(* Logix 5000 project; controller R5_CSS vendor 1 type 14 code 74 rev 19.11; software revision 19.01; part 8 of 20 *)
(* tags used below, declared in another part *)
   Const_CubicInchToGal : REAL;
   FC101 : FLOW_CONTROL;   // QUENCH BASIN FLOW TRANSMITTER CONTROL
   FC101_PIDE : PID_ENHANCED;
   FC140 : FLOW_CONTROL;
   FC140_DIFF_FT : REAL;
   FC140A : FLOW_CONTROL;   // QUENCH TOWER UPPER SPRAY FLOW CONTROL
   FC140A_FT_Pcnt : REAL;
   FC140B : FLOW_CONTROL;   // QUENCH TOWER LOWER SPRAY FLOW CONTROL
   FC140B_FT_Pcnt : REAL;
   FCV410 : ValveControl_TwoWay;
   FCV410_AUTO_ONS : BOOL;
   FCV410_ClosedMinSP : DINT;
   FCV410_ClosedTON : TIMER;
   FCV410_HoldDelaySecSP : DINT;
   FCV410_HoldDelayTOF : TIMER;
   FCV410_LT_Hold : BOOL;
   FCV410_MANUAL_ONS : BOOL;
   FCV410_On : BOOL;
   FCV410_Open : BOOL;
   FCV410_OpenSecSP : DINT;
   FCV410_OpenTON : TIMER;
   FireFlowAlarm_ONS2 : BOOL;
   FireFlowAlarm_SetLC101 : BOOL;
   FireFlowAlarmFromUTL : BOOL;
   FT140_Ratio : REAL;
   FT140_TOTAL_FLOW : REAL;
   H3_LC101 : LEVEL_CONTROL;
   HX401A : PUMP_CONTROL;   // HEAT EXCHANGER A
   HX401A_QI_AUTO_OS : BOOL;
   HX401A_QI_MAN_OS : BOOL;
   HX401B : PUMP_CONTROL;   // HEAT EXCHANGER B
   HX401B_QI_AUTO_OS : BOOL;
   HX401B_QI_MAN_OS : BOOL;
   LC101 : LEVEL_CONTROL;   // QUENCH TOWER BASIN LIT
   LC101_AUTO_ONS1 : BOOL;
   LC101_LAHH_MaxTime_TMR : TIMER;
   LC101_LAHH_MaxTimeAlm : BOOL;
   LC101_LAHH_MaxTimeMinSP : REAL;
   LC101_LT_Temp : REAL;
   LC101_MANUAL_ONS1 : BOOL;
   LC101_PIDE : PID_ENHANCED;
   LC101_PIDE_AUTO : BOOL;
   LC101_PIDE_CV_Hold : REAL;
   LC205 : LEVEL_CONTROL;   // OVERHEAD CONDENSER BASIN LEVEL CONTROL
   LC205_Totalize_Calc : BOOL;
   LC205_Totalize_End : REAL;
   LC205_Totalize_Gal : REAL;
   LC205_Totalize_Inches : REAL;
   LC205_Totalize_Ini : BOOL;
   LC205_Totalize_Start : REAL;
   LC205_Totalize_TOF : TIMER;
   LC205_Totalize_Vessel1_Diameter_inches : REAL;
   LC205_Totalize_Vessel1_Gal : REAL;
   LC205_Totalize_Vessel1_Rad_inches : REAL;
   LC205_Totalize_Vessel2_Diameter_inches : REAL;
   LC205_Totalize_Vessel2_Gal : REAL;
   LC205_Totalize_Vessel2_Rad_inches : REAL;
   LC303A : LEVEL_CONTROL;   // AQUEOUS PHASE OF PRIMARY SETTLER
   MV361 : ValveControl_TwoWay;
   MV361_AUTO_ONS1 : BOOL;
   MV361_Open : BOOL;
   ONE_SHOT : BOOL[32];
   P101A : PUMP_CONTROL;
   P101B : PUMP_CONTROL;
   P205 : PUMP_CONTROL;   // OVERHEAD CONDENSER TRANSFER PUMP
   P205_START_ONS : BOOL;
   P205_STOP_ONS : BOOL;
   PID1_TCV101 : PID;
   PID_TCV101_TON : TIMER;
   QuenchFlowMeterFailed : BOOL;
   TIMER : TIMER[50];   // HX A TIMER FOR START
   TMR_FAULT : DINT;
(* MainProgram, continued *)

ROUTINE FCV410_BasinLevelHotWaterFlushValve   (* ladder *)
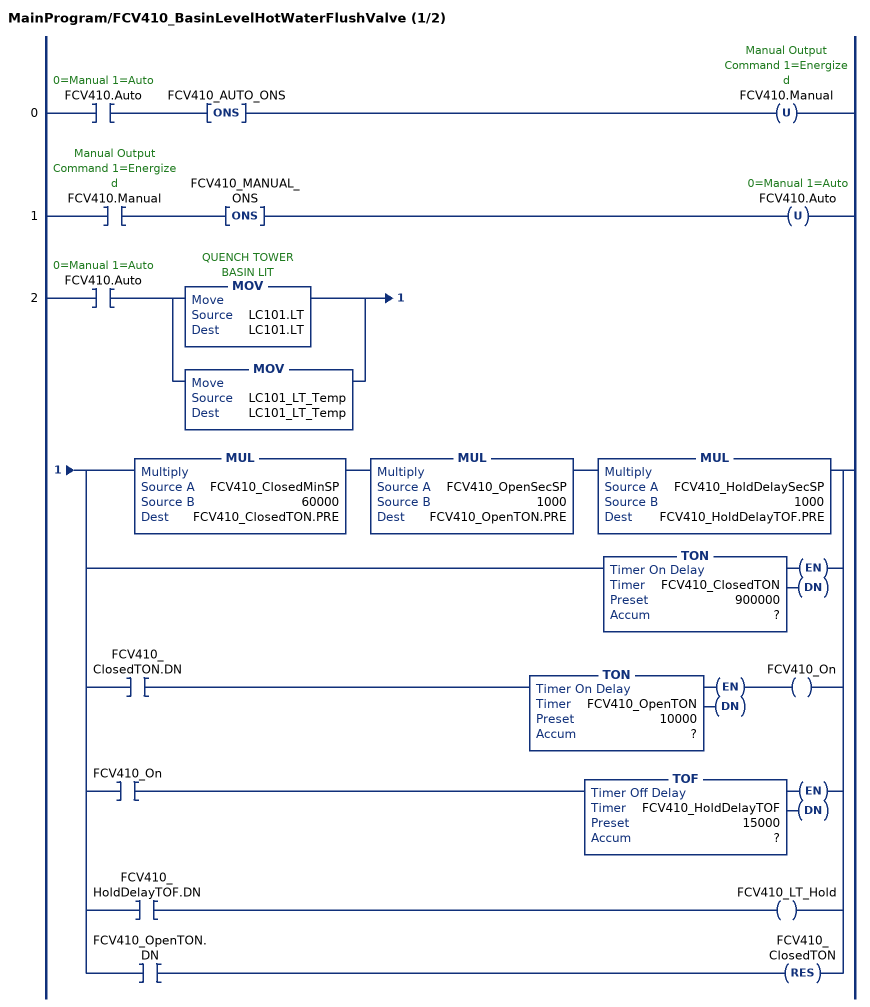
   0: XIC(FCV410.Auto)ONS(FCV410_AUTO_ONS)OTU(FCV410.Manual);
   1: XIC(FCV410.Manual)ONS(FCV410_MANUAL_ONS)OTU(FCV410.Auto);
   2: XIC(FCV410.Auto)[MOV(LC101.LT,LC101.LT) ,MOV(LC101_LT_Temp,LC101_LT_Temp) ][MUL(FCV410_ClosedMinSP,60000,FCV410_ClosedTON.PRE) MUL(FCV410_OpenSecSP,1000,FCV410_OpenTON.PRE) MUL(FCV410_HoldDelaySecSP,1000,FCV410_HoldDelayTOF.PRE) ,TON(FCV410_ClosedTON,?,?) ,XIC(FCV410_ClosedTON.DN) TON(FCV410_OpenTON,?,?) OTE(FCV410_On) ,XIC(FCV410_On) TOF(FCV410_HoldDelayTOF,?,?) ,XIC(FCV410_HoldDelayTOF.DN) OTE(FCV410_LT_Hold) ,XIC(FCV410_OpenTON.DN) RES(FCV410_ClosedTON) ];
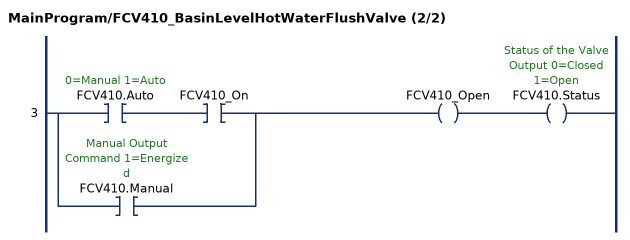
   3: [XIC(FCV410.Auto) XIC(FCV410_On) ,XIC(FCV410.Manual) ]OTE(FCV410_Open)OTE(FCV410.Status);
END_ROUTINE

ROUTINE FT140_QuenchFlowDelta   (* ladder *)
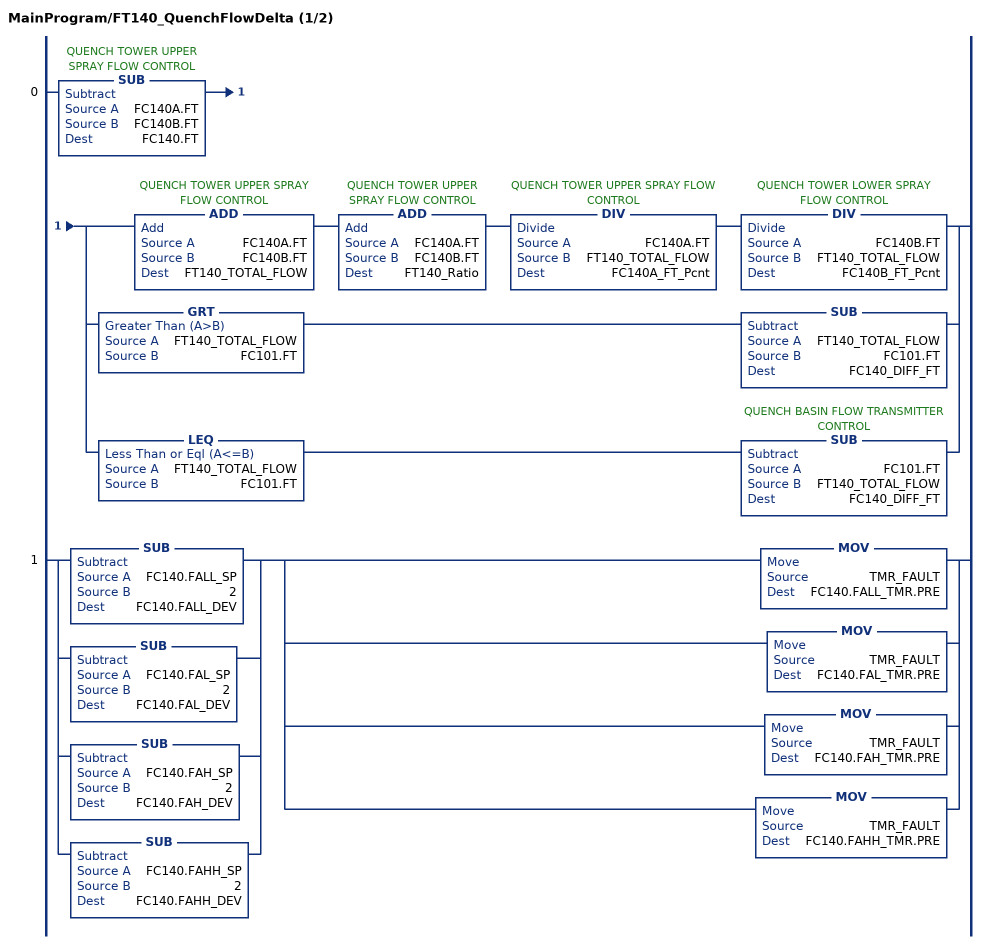
   0: SUB(FC140A.FT,FC140B.FT,FC140.FT)[ADD(FC140A.FT,FC140B.FT,FT140_TOTAL_FLOW) ADD(FC140A.FT,FC140B.FT,FT140_Ratio) DIV(FC140A.FT,FT140_TOTAL_FLOW,FC140A_FT_Pcnt) DIV(FC140B.FT,FT140_TOTAL_FLOW,FC140B_FT_Pcnt) ,GRT(FT140_TOTAL_FLOW,FC101.FT) SUB(FT140_TOTAL_FLOW,FC101.FT,FC140_DIFF_FT) ,LEQ(FT140_TOTAL_FLOW,FC101.FT) SUB(FC101.FT,FT140_TOTAL_FLOW,FC140_DIFF_FT) ];
   1: [SUB(FC140.FALL_SP,2,FC140.FALL_DEV) ,SUB(FC140.FAL_SP,2,FC140.FAL_DEV) ,SUB(FC140.FAH_SP,2,FC140.FAH_DEV) ,SUB(FC140.FAHH_SP,2,FC140.FAHH_DEV) ][MOV(TMR_FAULT,FC140.FALL_TMR.PRE) ,MOV(TMR_FAULT,FC140.FAL_TMR.PRE) ,MOV(TMR_FAULT,FC140.FAH_TMR.PRE) ,MOV(TMR_FAULT,FC140.FAHH_TMR.PRE) ];
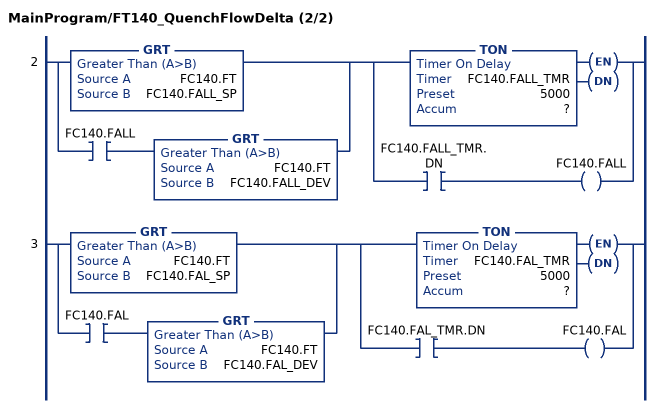
   2: [GRT(FC140.FT,FC140.FALL_SP) ,XIC(FC140.FALL) GRT(FC140.FT,FC140.FALL_DEV) ][TON(FC140.FALL_TMR,?,?) ,XIC(FC140.FALL_TMR.DN) OTE(FC140.FALL) ];
   3: [GRT(FC140.FT,FC140.FAL_SP) ,XIC(FC140.FAL) GRT(FC140.FT,FC140.FAL_DEV) ][TON(FC140.FAL_TMR,?,?) ,XIC(FC140.FAL_TMR.DN) OTE(FC140.FAL) ];
END_ROUTINE

ROUTINE HS361_T1_Occupancy_Valve   (* ladder *)
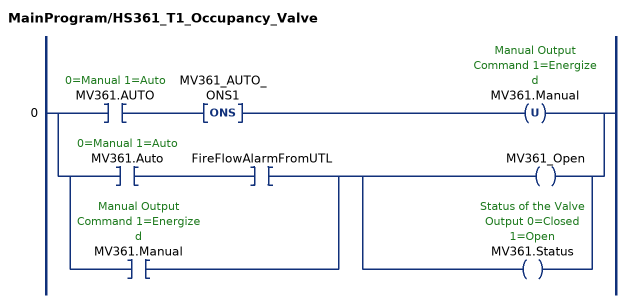
   0: [XIC(MV361.AUTO) ONS(MV361_AUTO_ONS1) OTU(MV361.Manual) ,[XIC(MV361.Auto) XIC(FireFlowAlarmFromUTL) ,XIC(MV361.Manual) ] [OTE(MV361_Open) ,OTE(MV361.Status) ] ];
END_ROUTINE

ROUTINE HX401A_HeatExchangerControl   (* ladder *)
// HEAT EXCHANGER 433
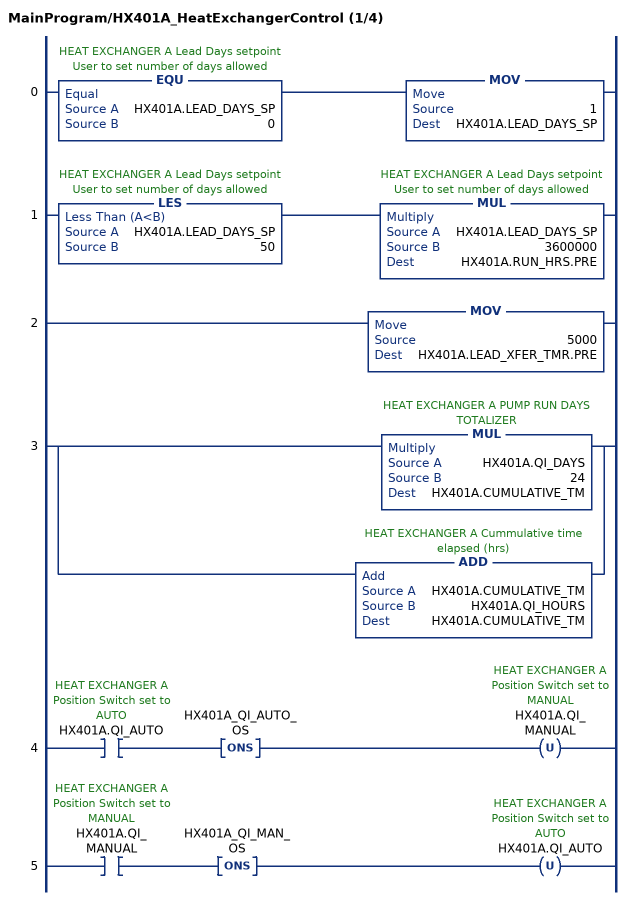
   0: EQU(HX401A.LEAD_DAYS_SP,0)MOV(1,HX401A.LEAD_DAYS_SP);
   1: LES(HX401A.LEAD_DAYS_SP,50)MUL(HX401A.LEAD_DAYS_SP,3600000,HX401A.RUN_HRS.PRE);
   2: MOV(5000,HX401A.LEAD_XFER_TMR.PRE);
   3: [MUL(HX401A.QI_DAYS,24,HX401A.CUMULATIVE_TM) ,ADD(HX401A.CUMULATIVE_TM,HX401A.QI_HOURS,HX401A.CUMULATIVE_TM) ];
   4: XIC(HX401A.QI_AUTO)ONS(HX401A_QI_AUTO_OS)OTU(HX401A.QI_MANUAL);
   5: XIC(HX401A.QI_MANUAL)ONS(HX401A_QI_MAN_OS)OTU(HX401A.QI_AUTO);
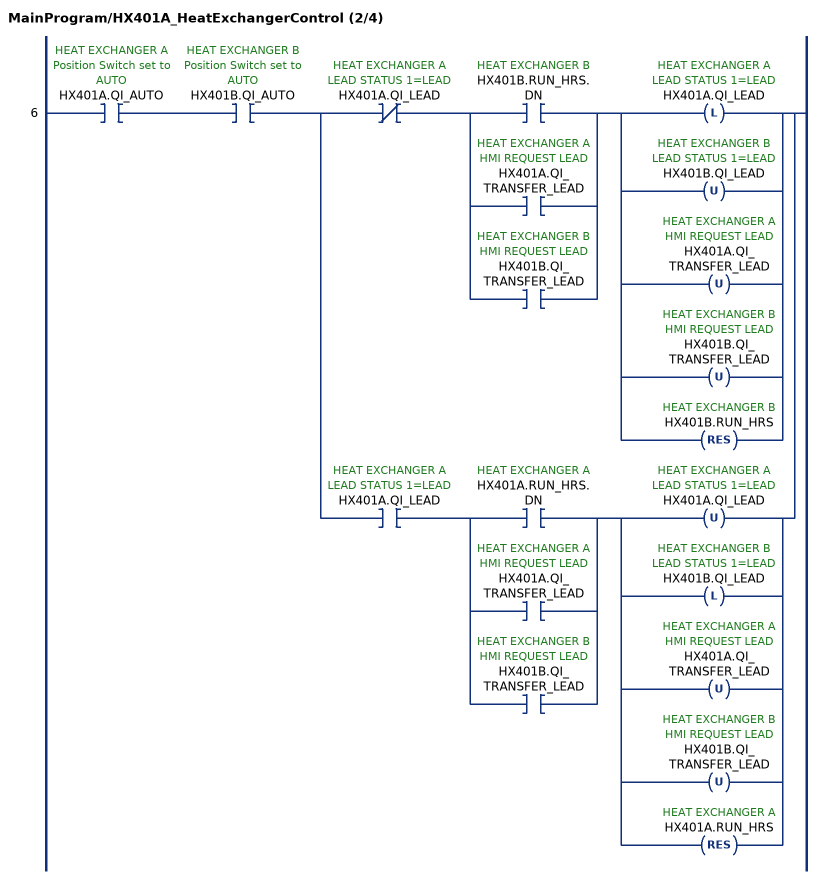
   6: XIC(HX401A.QI_AUTO)XIC(HX401B.QI_AUTO)[XIO(HX401A.QI_LEAD) [XIC(HX401B.RUN_HRS.DN) ,XIC(HX401A.QI_TRANSFER_LEAD) ,XIC(HX401B.QI_TRANSFER_LEAD) ] [OTL(HX401A.QI_LEAD) ,OTU(HX401B.QI_LEAD) ,OTU(HX401A.QI_TRANSFER_LEAD) ,OTU(HX401B.QI_TRANSFER_LEAD) ,RES(HX401B.RUN_HRS) ] ,XIC(HX401A.QI_LEAD) [XIC(HX401A.RUN_HRS.DN) ,XIC(HX401A.QI_TRANSFER_LEAD) ,XIC(HX401B.QI_TRANSFER_LEAD) ] [OTU(HX401A.QI_LEAD) ,OTL(HX401B.QI_LEAD) ,OTU(HX401A.QI_TRANSFER_LEAD) ,OTU(HX401B.QI_TRANSFER_LEAD) ,RES(HX401A.RUN_HRS) ] ];
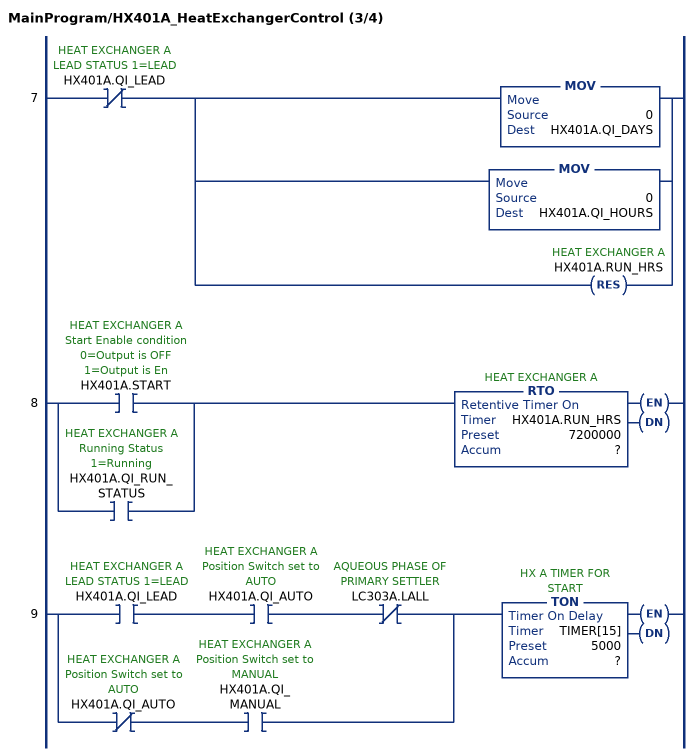
   7: XIO(HX401A.QI_LEAD)[MOV(0,HX401A.QI_DAYS) ,MOV(0,HX401A.QI_HOURS) ,RES(HX401A.RUN_HRS) ];
   8: [XIC(HX401A.START) ,XIC(HX401A.QI_RUN_STATUS) ]RTO(HX401A.RUN_HRS,?,?);
   9: [XIC(HX401A.QI_LEAD) XIC(HX401A.QI_AUTO) XIO(LC303A.LALL) ,XIO(HX401A.QI_AUTO) XIC(HX401A.QI_MANUAL) ]TON(TIMER[15],?,?);
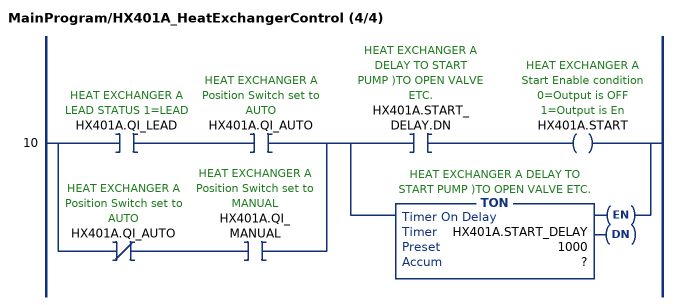
   10: [XIC(HX401A.QI_LEAD) XIC(HX401A.QI_AUTO) ,XIO(HX401A.QI_AUTO) XIC(HX401A.QI_MANUAL) ][XIC(HX401A.START_DELAY.DN) OTE(HX401A.START) ,TON(HX401A.START_DELAY,?,?) ];
END_ROUTINE

ROUTINE HX401B_HeatExchangerControl   (* ladder *)
// HEAT EXCHANGER 433
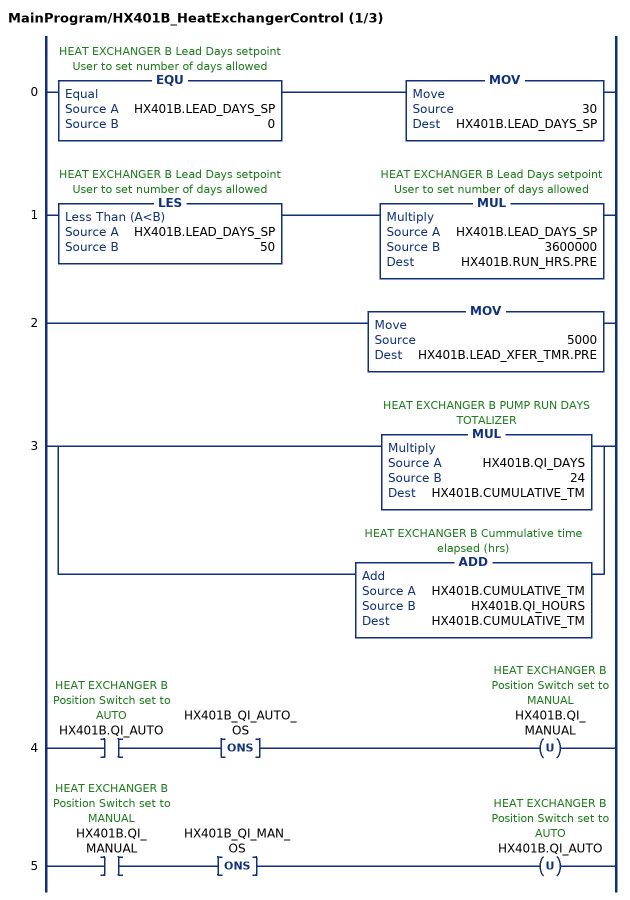
   0: EQU(HX401B.LEAD_DAYS_SP,0)MOV(30,HX401B.LEAD_DAYS_SP);
   1: LES(HX401B.LEAD_DAYS_SP,50)MUL(HX401B.LEAD_DAYS_SP,3600000,HX401B.RUN_HRS.PRE);
   2: MOV(5000,HX401B.LEAD_XFER_TMR.PRE);
   3: [MUL(HX401B.QI_DAYS,24,HX401B.CUMULATIVE_TM) ,ADD(HX401B.CUMULATIVE_TM,HX401B.QI_HOURS,HX401B.CUMULATIVE_TM) ];
   4: XIC(HX401B.QI_AUTO)ONS(HX401B_QI_AUTO_OS)OTU(HX401B.QI_MANUAL);
   5: XIC(HX401B.QI_MANUAL)ONS(HX401B_QI_MAN_OS)OTU(HX401B.QI_AUTO);
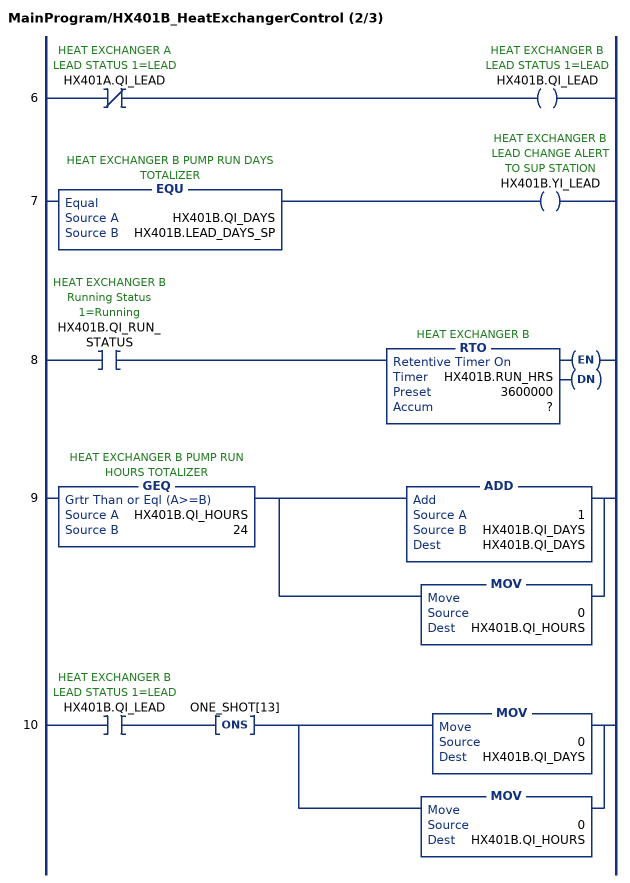
   6: XIO(HX401A.QI_LEAD)OTE(HX401B.QI_LEAD);
   7: EQU(HX401B.QI_DAYS,HX401B.LEAD_DAYS_SP)OTE(HX401B.YI_LEAD);
   8: XIC(HX401B.QI_RUN_STATUS)RTO(HX401B.RUN_HRS,?,?);
   9: GEQ(HX401B.QI_HOURS,24)[ADD(1,HX401B.QI_DAYS,HX401B.QI_DAYS) ,MOV(0,HX401B.QI_HOURS) ];
   10: XIC(HX401B.QI_LEAD)ONS(ONE_SHOT[13])[MOV(0,HX401B.QI_DAYS) ,MOV(0,HX401B.QI_HOURS) ];
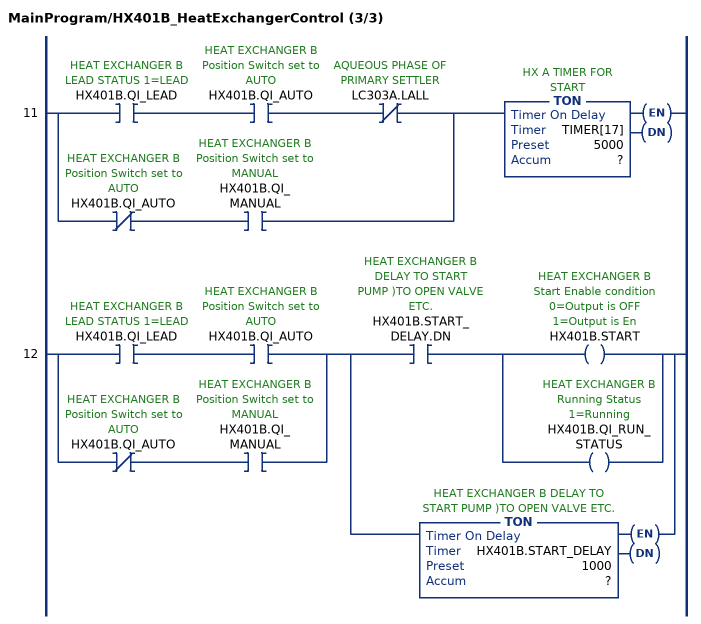
   11: [XIC(HX401B.QI_LEAD) XIC(HX401B.QI_AUTO) XIO(LC303A.LALL) ,XIO(HX401B.QI_AUTO) XIC(HX401B.QI_MANUAL) ]TON(TIMER[17],?,?);
   12: [XIC(HX401B.QI_LEAD) XIC(HX401B.QI_AUTO) ,XIO(HX401B.QI_AUTO) XIC(HX401B.QI_MANUAL) ][XIC(HX401B.START_DELAY.DN) [OTE(HX401B.START) ,OTE(HX401B.QI_RUN_STATUS) ] ,TON(HX401B.START_DELAY,?,?) ];
END_ROUTINE

ROUTINE LC101_BasinLevel_PID   (* ladder *)
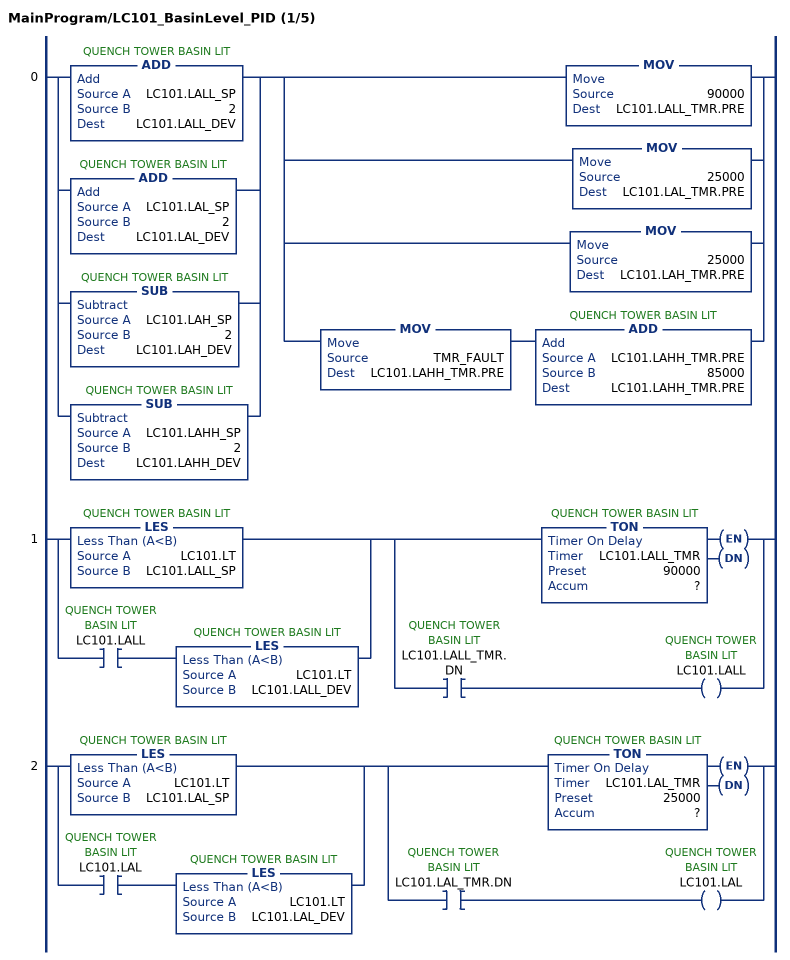
   0: [ADD(LC101.LALL_SP,2,LC101.LALL_DEV) ,ADD(LC101.LAL_SP,2,LC101.LAL_DEV) ,SUB(LC101.LAH_SP,2,LC101.LAH_DEV) ,SUB(LC101.LAHH_SP,2,LC101.LAHH_DEV) ][MOV(90000,LC101.LALL_TMR.PRE) ,MOV(25000,LC101.LAL_TMR.PRE) ,MOV(25000,LC101.LAH_TMR.PRE) ,MOV(TMR_FAULT,LC101.LAHH_TMR.PRE) ADD(LC101.LAHH_TMR.PRE,85000,LC101.LAHH_TMR.PRE) ];
   1: [LES(LC101.LT,LC101.LALL_SP) ,XIC(LC101.LALL) LES(LC101.LT,LC101.LALL_DEV) ][TON(LC101.LALL_TMR,?,?) ,XIC(LC101.LALL_TMR.DN) OTE(LC101.LALL) ];
   2: [LES(LC101.LT,LC101.LAL_SP) ,XIC(LC101.LAL) LES(LC101.LT,LC101.LAL_DEV) ][TON(LC101.LAL_TMR,?,?) ,XIC(LC101.LAL_TMR.DN) OTE(LC101.LAL) ];
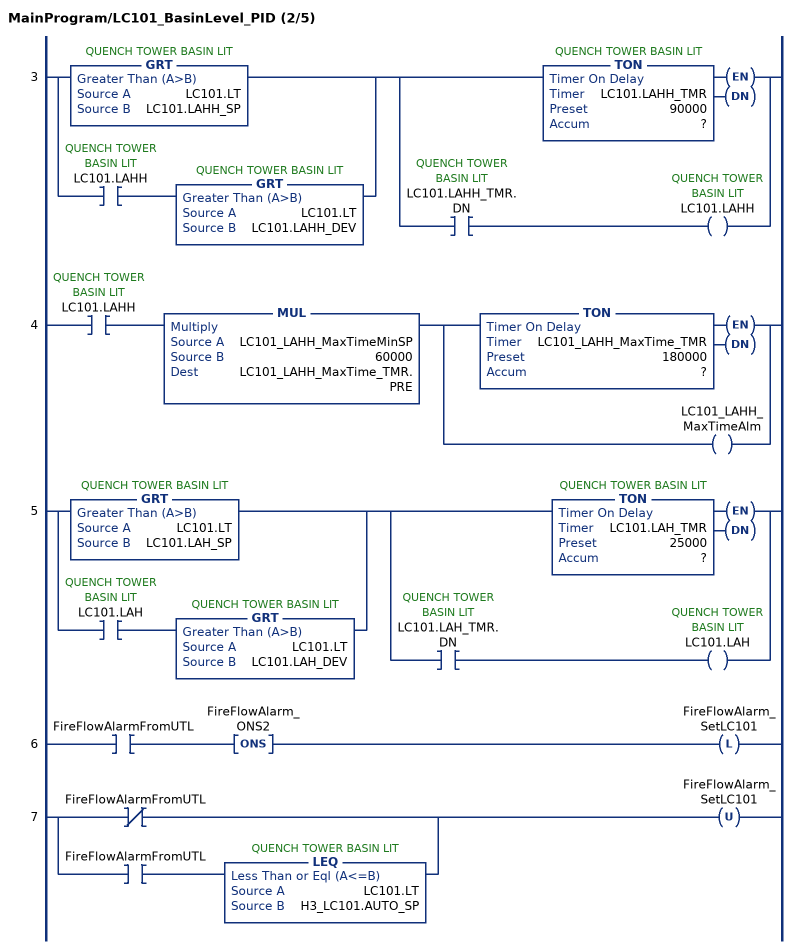
   3: [GRT(LC101.LT,LC101.LAHH_SP) ,XIC(LC101.LAHH) GRT(LC101.LT,LC101.LAHH_DEV) ][TON(LC101.LAHH_TMR,?,?) ,XIC(LC101.LAHH_TMR.DN) OTE(LC101.LAHH) ];
   4: XIC(LC101.LAHH)MUL(LC101_LAHH_MaxTimeMinSP,60000,LC101_LAHH_MaxTime_TMR.PRE)[TON(LC101_LAHH_MaxTime_TMR,?,?) ,OTE(LC101_LAHH_MaxTimeAlm) ];
   5: [GRT(LC101.LT,LC101.LAH_SP) ,XIC(LC101.LAH) GRT(LC101.LT,LC101.LAH_DEV) ][TON(LC101.LAH_TMR,?,?) ,XIC(LC101.LAH_TMR.DN) OTE(LC101.LAH) ];
   6: XIC(FireFlowAlarmFromUTL)ONS(FireFlowAlarm_ONS2)OTL(FireFlowAlarm_SetLC101);
   7: [XIO(FireFlowAlarmFromUTL) ,XIC(FireFlowAlarmFromUTL) LEQ(LC101.LT,H3_LC101.AUTO_SP) ]OTU(FireFlowAlarm_SetLC101);
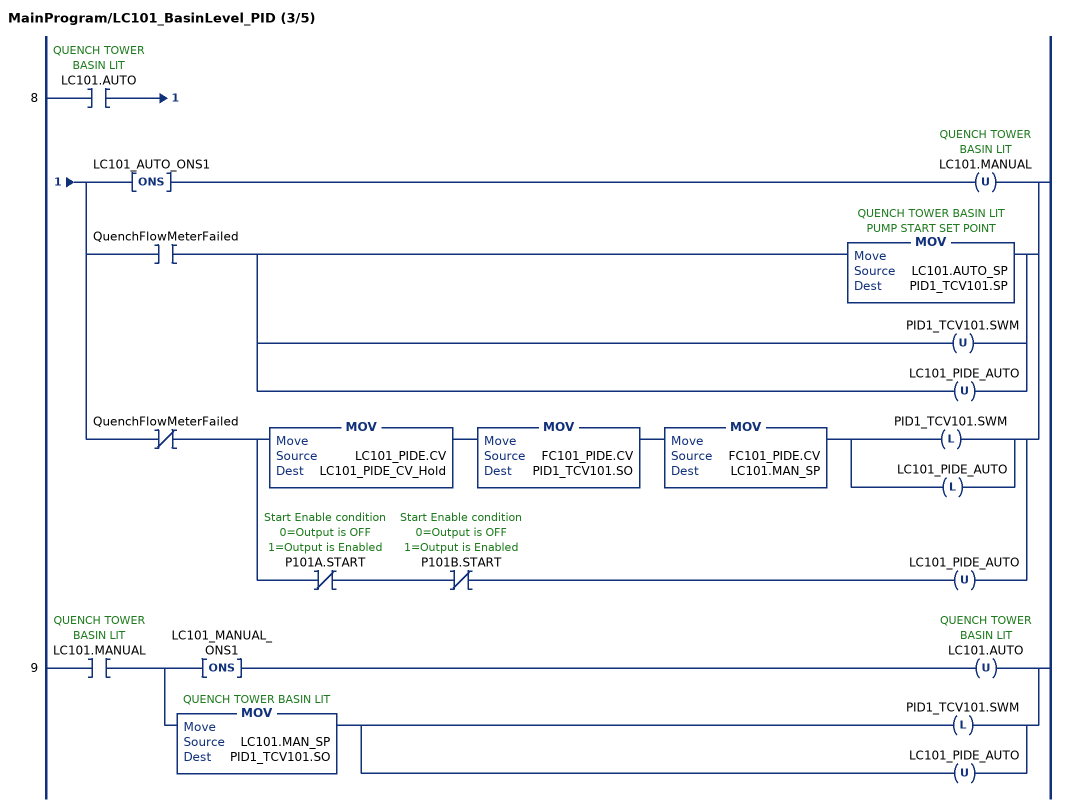
   8: XIC(LC101.AUTO)[ONS(LC101_AUTO_ONS1) OTU(LC101.MANUAL) ,XIC(QuenchFlowMeterFailed) [MOV(LC101.AUTO_SP,PID1_TCV101.SP) ,OTU(PID1_TCV101.SWM) ,OTU(LC101_PIDE_AUTO) ] ,XIO(QuenchFlowMeterFailed) [MOV(LC101_PIDE.CV,LC101_PIDE_CV_Hold) MOV(FC101_PIDE.CV,PID1_TCV101.SO) MOV(FC101_PIDE.CV,LC101.MAN_SP) [OTL(PID1_TCV101.SWM) ,OTL(LC101_PIDE_AUTO) ] ,XIO(P101A.START) XIO(P101B.START) OTU(LC101_PIDE_AUTO) ] ];
   9: XIC(LC101.MANUAL)[ONS(LC101_MANUAL_ONS1) OTU(LC101.AUTO) ,MOV(LC101.MAN_SP,PID1_TCV101.SO) [OTL(PID1_TCV101.SWM) ,OTU(LC101_PIDE_AUTO) ] ];
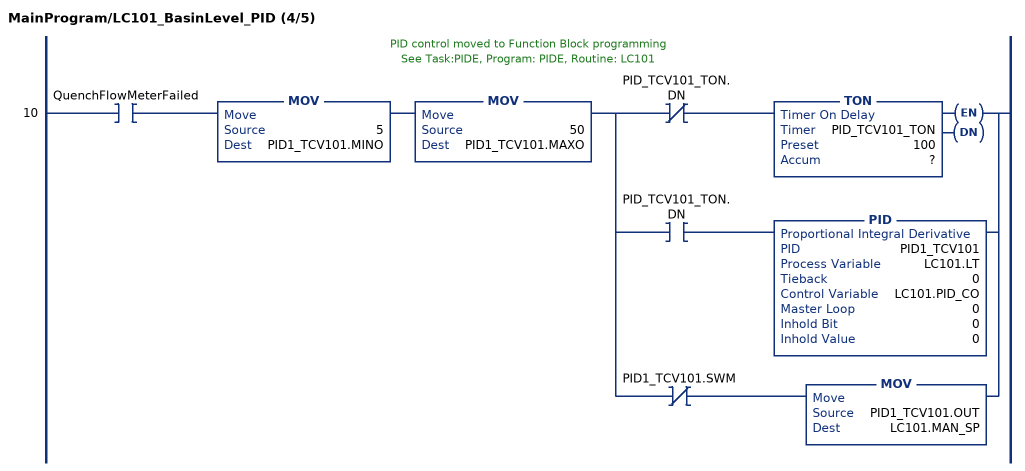
   // PID control moved to Function Block programming
   // See Task:PIDE, Program: PIDE, Routine: LC101
   10: XIC(QuenchFlowMeterFailed)MOV(5,PID1_TCV101.MINO)MOV(50,PID1_TCV101.MAXO)[XIO(PID_TCV101_TON.DN) TON(PID_TCV101_TON,?,?) ,XIC(PID_TCV101_TON.DN) PID(PID1_TCV101,LC101.LT,0,LC101.PID_CO,0,0,0) ,XIO(PID1_TCV101.SWM) MOV(PID1_TCV101.OUT,LC101.MAN_SP) ];
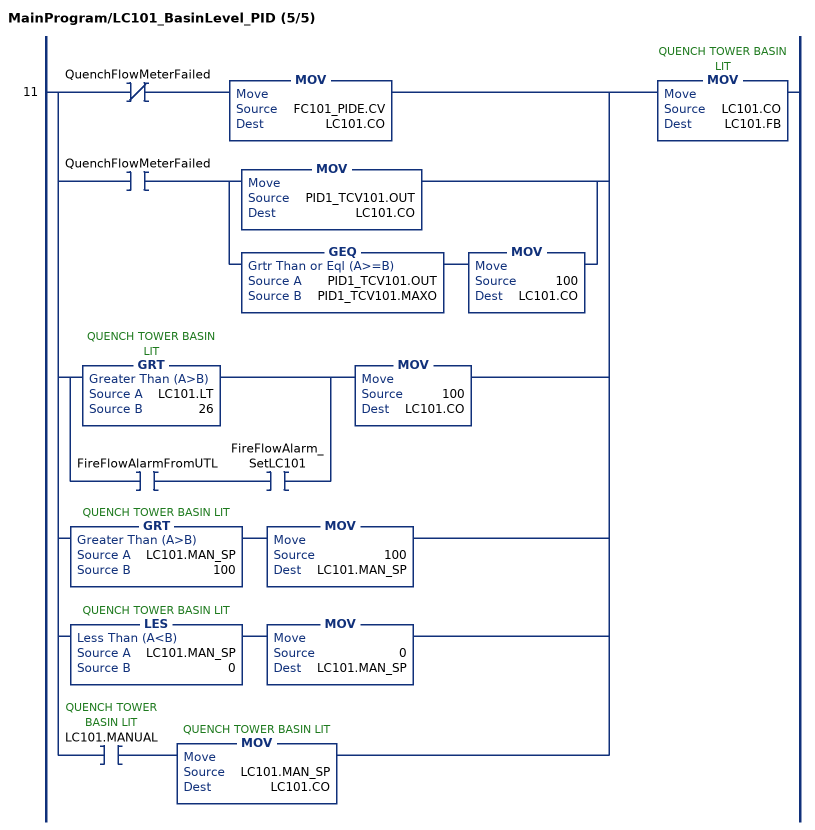
   11: [XIO(QuenchFlowMeterFailed) MOV(FC101_PIDE.CV,LC101.CO) ,XIC(QuenchFlowMeterFailed) [MOV(PID1_TCV101.OUT,LC101.CO) ,GEQ(PID1_TCV101.OUT,PID1_TCV101.MAXO) MOV(100,LC101.CO) ] ,[GRT(LC101.LT,26) ,XIC(FireFlowAlarmFromUTL) XIC(FireFlowAlarm_SetLC101) ] MOV(100,LC101.CO) ,GRT(LC101.MAN_SP,100) MOV(100,LC101.MAN_SP) ,LES(LC101.MAN_SP,0) MOV(0,LC101.MAN_SP) ,XIC(LC101.MANUAL) MOV(LC101.MAN_SP,LC101.CO) ]MOV(LC101.CO,LC101.FB);
END_ROUTINE

ROUTINE LC205_OverheadCondBasinLevel   (* ladder *)
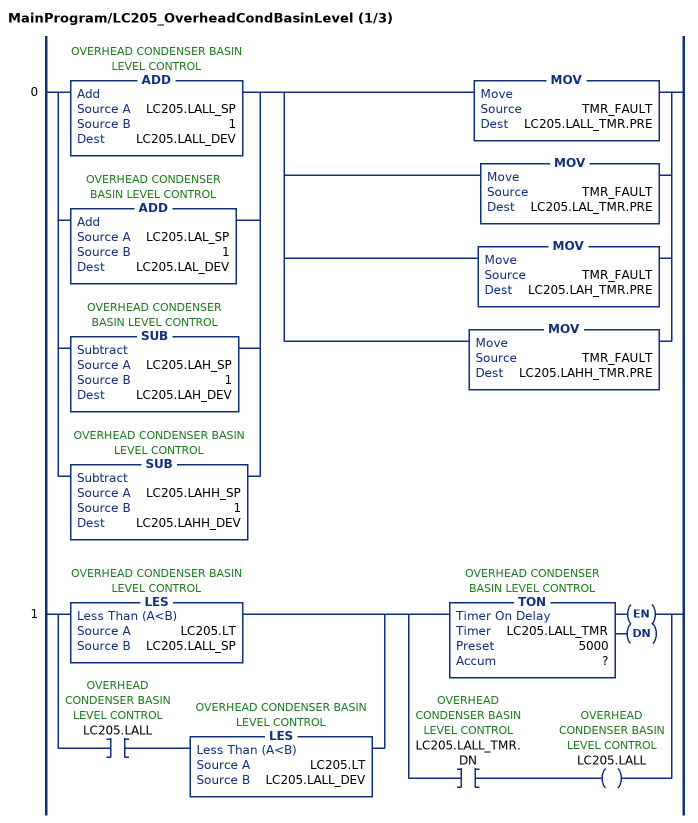
   0: [ADD(LC205.LALL_SP,1,LC205.LALL_DEV) ,ADD(LC205.LAL_SP,1,LC205.LAL_DEV) ,SUB(LC205.LAH_SP,1,LC205.LAH_DEV) ,SUB(LC205.LAHH_SP,1,LC205.LAHH_DEV) ][MOV(TMR_FAULT,LC205.LALL_TMR.PRE) ,MOV(TMR_FAULT,LC205.LAL_TMR.PRE) ,MOV(TMR_FAULT,LC205.LAH_TMR.PRE) ,MOV(TMR_FAULT,LC205.LAHH_TMR.PRE) ];
   1: [LES(LC205.LT,LC205.LALL_SP) ,XIC(LC205.LALL) LES(LC205.LT,LC205.LALL_DEV) ][TON(LC205.LALL_TMR,?,?) ,XIC(LC205.LALL_TMR.DN) OTE(LC205.LALL) ];
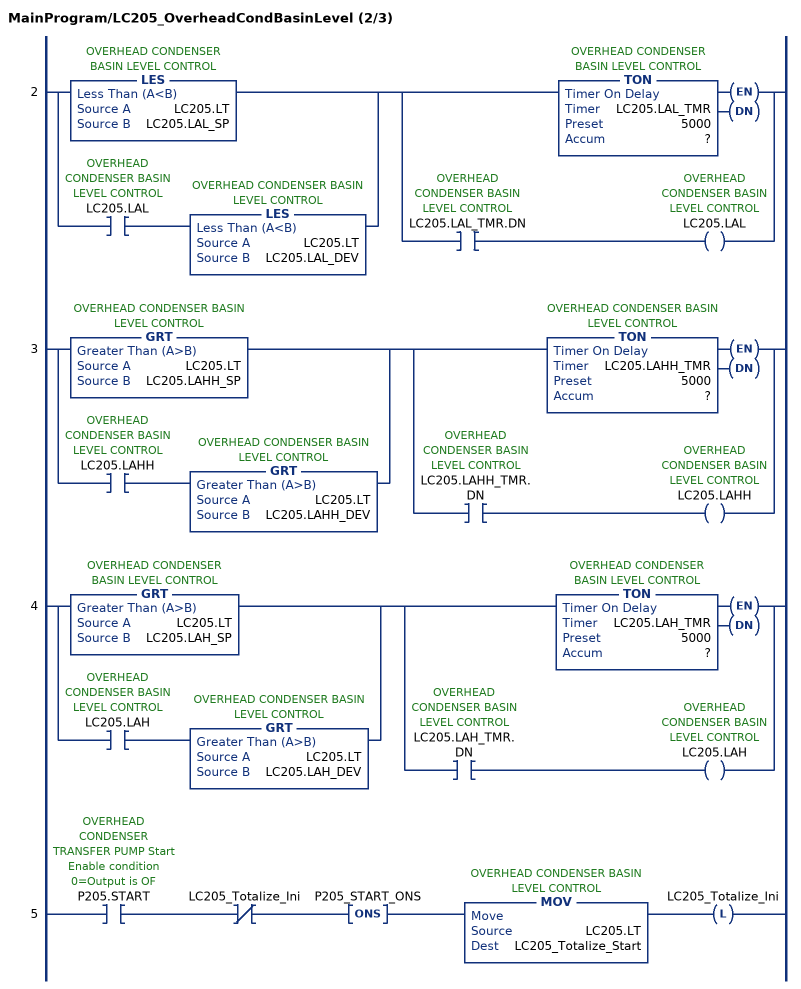
   2: [LES(LC205.LT,LC205.LAL_SP) ,XIC(LC205.LAL) LES(LC205.LT,LC205.LAL_DEV) ][TON(LC205.LAL_TMR,?,?) ,XIC(LC205.LAL_TMR.DN) OTE(LC205.LAL) ];
   3: [GRT(LC205.LT,LC205.LAHH_SP) ,XIC(LC205.LAHH) GRT(LC205.LT,LC205.LAHH_DEV) ][TON(LC205.LAHH_TMR,?,?) ,XIC(LC205.LAHH_TMR.DN) OTE(LC205.LAHH) ];
   4: [GRT(LC205.LT,LC205.LAH_SP) ,XIC(LC205.LAH) GRT(LC205.LT,LC205.LAH_DEV) ][TON(LC205.LAH_TMR,?,?) ,XIC(LC205.LAH_TMR.DN) OTE(LC205.LAH) ];
   5: XIC(P205.START)XIO(LC205_Totalize_Ini)ONS(P205_START_ONS)MOV(LC205.LT,LC205_Totalize_Start)OTL(LC205_Totalize_Ini);
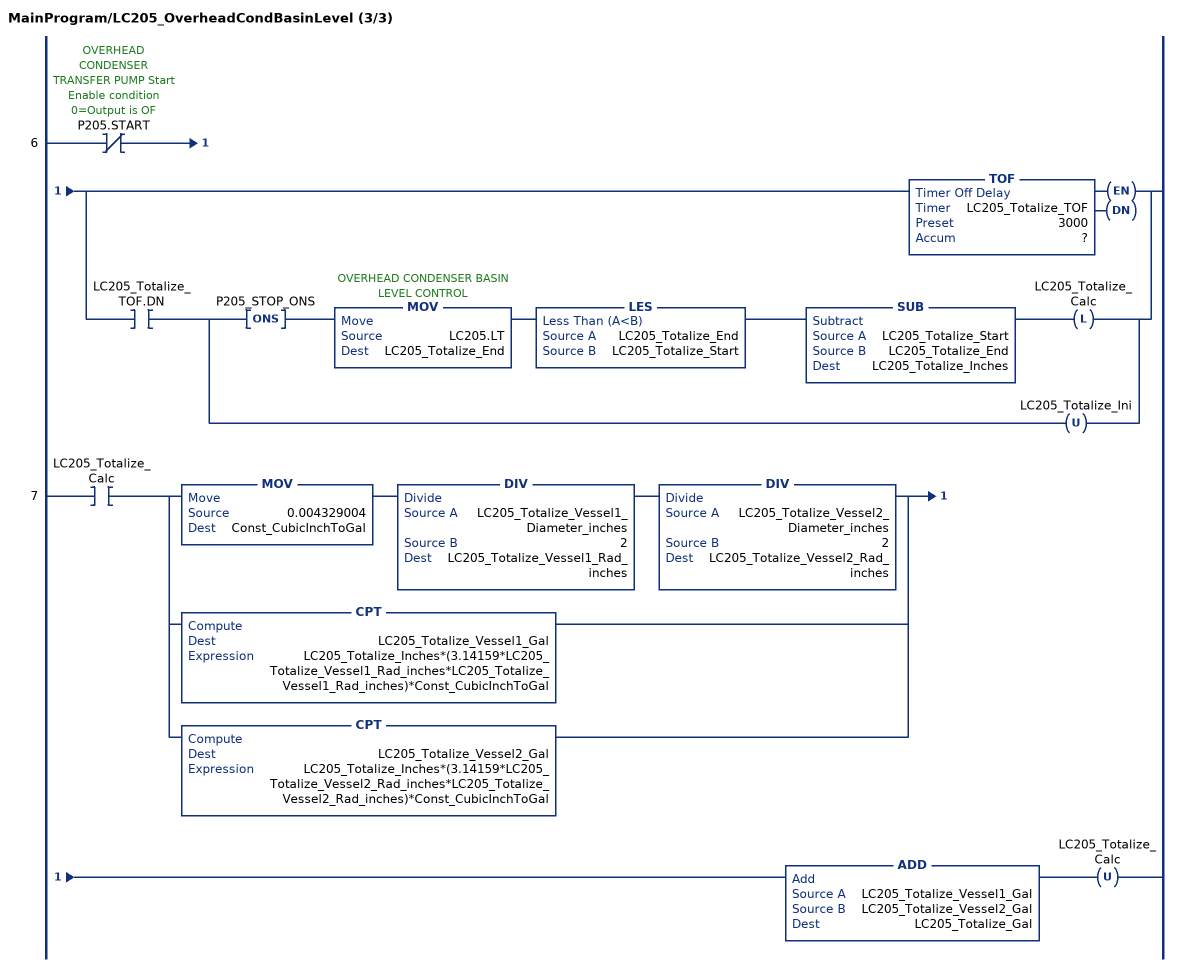
   6: XIO(P205.START)[TOF(LC205_Totalize_TOF,?,?) ,XIC(LC205_Totalize_TOF.DN) [ONS(P205_STOP_ONS) MOV(LC205.LT,LC205_Totalize_End) LES(LC205_Totalize_End,LC205_Totalize_Start) SUB(LC205_Totalize_Start,LC205_Totalize_End,LC205_Totalize_Inches) OTL(LC205_Totalize_Calc) ,OTU(LC205_Totalize_Ini) ] ];
   7: XIC(LC205_Totalize_Calc)[MOV(0.004329004,Const_CubicInchToGal) DIV(LC205_Totalize_Vessel1_Diameter_inches,2,LC205_Totalize_Vessel1_Rad_inches) DIV(LC205_Totalize_Vessel2_Diameter_inches,2,LC205_Totalize_Vessel2_Rad_inches) ,CPT(LC205_Totalize_Vessel1_Gal,LC205_Totalize_Inches*(3.14159*LC205_Totalize_Vessel1_Rad_inches*LC205_Totalize_Vessel1_Rad_inches)*Const_CubicInchToGal) ,CPT(LC205_Totalize_Vessel2_Gal,LC205_Totalize_Inches*(3.14159*LC205_Totalize_Vessel2_Rad_inches*LC205_Totalize_Vessel2_Rad_inches)*Const_CubicInchToGal) ]ADD(LC205_Totalize_Vessel1_Gal,LC205_Totalize_Vessel2_Gal,LC205_Totalize_Gal)OTU(LC205_Totalize_Calc);
END_ROUTINE
